TEXTLIST AxisState_txt
  0 = 'INVALID'
  1 = 'DISABLED'
  2 = 'STANDSTILL'
  3 = 'ERROR STOP'
  4 = 'STOPPING'
  5 = 'HOMING'
  6 = 'DISCRETE MOTION'
  7 = 'CONTINIOUS MOTION'
  8 = 'SYNCHRONIZED MOTION'
   = ''
END_TEXTLIST

(* stored: Version 1.1.0.1, ProductVersion 3.1.4024.11
   TextList AxisState_txt: Id {58d6d1b2-edaa-407b-9054-2e2edb62a1a4} *)
